FUNCTION_BLOCK INTERNAL FINAL FB_TestWrongSizeMessage IMPLEMENTS I_Message
VAR
    fbMessageParser : FB_MessageParser(ipMessage:= THIS^);
    fbMessageWriter : FB_MessageWriter(ipMessage:= THIS^);
    nValue : UDINT := 16#12345678;
END_VAR

METHOD CalculateSize : UDINT
VAR_INPUT
END_VAR
CalculateSize := 0;
END_METHOD

METHOD MergeFrom : HRESULT
VAR_IN_OUT
    fbParseCtx : FB_ParseContext;
END_VAR
VAR
    nTag : UDINT;
END_VAR
REPEAT
MergeFrom := fbParseCtx.ReadTag(nTag=> nTag);
IF SUCCEEDED(MergeFrom) AND nTag = 0 THEN
    EXIT;
END_IF

IF FAILED(MergeFrom) THEN
    RETURN;
END_IF

CASE nTag OF
    16#0D:
        MergeFrom := fbParseCtx.ReadFixed32(nValue=> nValue);
ELSE
    MergeFrom := fbParseCtx.SkipLastField();
END_CASE
UNTIL FAILED(MergeFrom) OR nTag = 0
END_REPEAT
END_METHOD

PROPERTY MessageValue : T_Any
GET
MessageValue := F_ToAnyType(anyArg:= nValue);
END_GET
END_PROPERTY

PROPERTY Parser : REFERENCE TO FB_MessageParser
GET
Parser REF= fbMessageParser;
END_GET
END_PROPERTY

PROPERTY Writer : REFERENCE TO FB_MessageWriter
GET
Writer REF= fbMessageWriter;
END_GET
END_PROPERTY

METHOD WriteTo : HRESULT
VAR_IN_OUT
    fbWriteCtx : FB_WriteContext;
END_VAR
WriteTo := fbWriteCtx.WriteTag(1, E_WireType.Fixed32);
IF FAILED(WriteTo) THEN
    RETURN;
END_IF

WriteTo := fbWriteCtx.WriteFixed32(nValue);
END_METHOD

END_FUNCTION_BLOCK

(* stored: Version 1.1.0.1
   POU FB_TestWrongSizeMessage: Id {2b68e746-e12d-4b21-925f-5d7e0bfc8565}, SpecialFunc None
   Method CalculateSize: Id {a85863f3-4cf4-4769-9ba2-c7d3a5c3d91e}
   Method MergeFrom: Id {22ce2046-bc8b-4cf7-9a19-0cdd55d4a9f4}
   Property MessageValue: Id {4db8ad67-0874-4de4-91dd-056892758087}
   Get Get: Id {bfa95f03-fc05-4823-a770-b5085691588c}
   Property Parser: Id {7cc7a907-9f3c-49a6-8aae-6bb014739329}
   Get Get: Id {8e432687-e78d-4ffb-8df0-f4ed5115d4a4}
   Property Writer: Id {0ec71936-2ff8-4033-8cbb-0d0a7bfca3eb}
   Get Get: Id {d2244500-cd5a-4275-be41-079d34c88e98}
   Method WriteTo: Id {0eecf5d0-6d38-4688-ae00-12eb077cf345} *)
